GLOBALCONSTANTS AuxiliaryState (* Value of auxiliary inputs constants *)
  (* Standard: 61499-1; Description: Copyright (c) 2024 HR Agrartechnik GmbH This program and the accompanying materials are made available under the terms of the Eclipse Public License 2.0 which is available at https://www.eclipse.org/legal/epl-2.0/ SPDX-License-Identifier: EPL-2.0 *)
  (* Version 1.0, 2024-01-25, Franz Höpfinger, HR Agrartechnik GmbH *)
  PACKAGE isobus::UT::io::Auxiliary::IN;
  VAR_GLOBAL CONSTANT
    AuxDisabled : isobus::UT::io::Auxiliary::IN::AuxiliaryState_S := (value := 0); (* Off - backward, down, left, or not pressed *)
    AuxDisabled_START : isobus::UT::io::Auxiliary::IN::AuxiliaryState_S := (value := 0, bCyclic := FALSE); (* Off - backward, down, left, or not pressed *)
    AuxEnabled : isobus::UT::io::Auxiliary::IN::AuxiliaryState_S := (value := 1); (* On  - forward, up, right, or pressed *)
    AuxEnabled_START : isobus::UT::io::Auxiliary::IN::AuxiliaryState_S := (value := 1, bCyclic := FALSE); (* On  - forward, up, right, or pressed *)
    AuxHeld : isobus::UT::io::Auxiliary::IN::AuxiliaryState_S := (value := 2); (* Held (forward, up, or right) *)
    AuxHeld_START : isobus::UT::io::Auxiliary::IN::AuxiliaryState_S := (value := 2, bCyclic := FALSE); (* Held (forward, up, or right) *)
    AuxEnabledBackwards : isobus::UT::io::Auxiliary::IN::AuxiliaryState_S := (value := 4); (* On momentary - backward, down or left *)
    AuxHeldBackwards : isobus::UT::io::Auxiliary::IN::AuxiliaryState_S := (value := 8); (* Held (backwards, down, or left) *)
    AuxHeldBackwards_START : isobus::UT::io::Auxiliary::IN::AuxiliaryState_S := (value := 8, bCyclic := FALSE); (* Held (backwards, down, or left) *)
    AuxDefault : isobus::UT::io::Auxiliary::IN::AuxiliaryState_S := (value := 9); (* - *)
    Invalid : isobus::UT::io::Auxiliary::IN::AuxiliaryState_S := (value := 255);
  END_VAR
END_GLOBALCONSTANTS
